{attribute 'linkalways'} 
{attribute 'no_explicit_call' := 'This FB is a CLASS and must be accessed using methods or properties'}
{attribute 'enable_dynamic_creation'}
FUNCTION_BLOCK MockBasicDigitalInput EXTENDS BasicDigitalInput

METHOD MockSetRawInputFalse : BOOL
SUPER^.input := FALSE;
END_METHOD

METHOD MockSetRawInputTrue : BOOL
SUPER^.input := TRUE;
END_METHOD

END_FUNCTION_BLOCK

(* stored: Version 1.1.0.1, ProductVersion 3.1.4024.12
   POU MockBasicDigitalInput: Id {11cf0b6b-9b3e-486d-ae9d-ca79f84cd47f}, SpecialFunc None
   Method MockSetRawInputFalse: Id {e789ecae-a502-0ace-02ca-972502205f00}
   Method MockSetRawInputTrue: Id {219cc62b-c677-017e-204e-0279319c58cf} *)
